Staubli VAL3: save.pgx

public program save()
// save the process list
  local num i
begin
  // setMutex
  setMutex(cycleStatus:bMutex)
  // save IT
  if saveCycle:libSave()!=0
    delay(0.5)
    i=saveCycle:libSave()
    if i!=0
      popUpMsg("libsave cycle error: "+toString("",i))
      logMsg("[KERNEL] CYCLE:Error saving cycle "+toString("",i))
    endIf
  endIf
  //release
  cycleStatus:bMutex=false
end
